TYPE ST_CoeParameter :
STRUCT
	nValue : BYTE;
	nIndex : WORD;
	nSubIndex : BYTE;
END_STRUCT
END_TYPE

(* stored: Version 1.1.0.1, ProductVersion 3.1.4022.18
   DUT ST_CoeParameter: Id {d0d0df25-ee6f-45b4-9851-a5ed58c99a79} *)
